// TIA Portal V17 export
// export: Created 2026-04-13T11:12:43.2975863Z, ExportSetting WithDefaults, DisplayName Totally Integrated Automation Portal, DisplayVersion V17 Update 4, DisplayName TIA Portal Openness, DisplayVersion V17 Update 4, DisplayName TIA Portal Version Control Interface, DisplayVersion V17, DisplayName SINAMICS Startdrive Advanced, DisplayVersion V17, DisplayName SINAMICS Startdrive G130, G150, S120, S150, SINAMICS MV, S210, DisplayVersion V17, DisplayName SINAMICS Startdrive G110M, G120, G120C, G120D, G120P, G115D, DisplayVersion V17, DisplayName STEP 7 Professional, DisplayVersion V17 Update 4, DisplayName STEP 7 Safety, DisplayVersion V17, DisplayName WinCC Professional, DisplayVersion V17 Update 4
FUNCTION "Byte数组_to_INT" : Void   // FC52, SCL
{ S7_Optimized_Access := 'TRUE' }
VERSION : 0.1
// stored: AutoNumber false, IsIECCheckEnabled false, SetENOAutomatically false, UDAEnableTagReadback false
   VAR_INPUT
      byte数组 : Array[*] of Byte;
      起始偏置 : Int;   // 从数组的第偏置位开始
   END_VAR
   VAR_OUTPUT
      "INT" : Int;
   END_VAR
   VAR_TEMP
      temp_int : Int;
   END_VAR
BEGIN

   #temp_int:=BYTE_TO_INT(#byte数组[#起始偏置]);
   #INT := SHL(IN := #temp_int, N := 8) + #byte数组[#起始偏置 + 1];
END_FUNCTION
